(*

.. <legal notes>

legal notes
=================
| SPDX-FileCopyrightText: © 2026 Oleksandr Tiutyk <trofimich@gmail.com>
| SPDX-License-Identifier: LGPL-3.0-only
| For details check: LGPL-3.0-only_

.. _LGPL-3.0-only: https://www.gnu.org/licenses/lgpl-3.0.en.html

.. </legal notes>

*)

{attribute 'no_explicit_call' := 'do not call this function block directly'} 
FUNCTION_BLOCK AdsLogger EXTENDS Object IMPLEMENTS ILogger
VAR
	_ClassName : STRING := __POUNAME();
END_VAR

{attribute 'monitoring' := 'call'}
PROPERTY ClassName : REFERENCE TO STRING
GET
ClassName REF= _ClassName;
END_GET
END_PROPERTY

METHOD Execute
// nothing to do for ADS logger
END_METHOD

{attribute 'monitoring' := 'call'}
PROPERTY NamespaceName : STRING
GET
NamespaceName := CurrentNamespace.Name;
END_GET
END_PROPERTY

{attribute 'monitoring' := 'call'}
PROPERTY SelfSize : ULINT
GET
SelfSize := XSIZEOF(THIS^);
END_GET
END_PROPERTY

METHOD TryLogError : BOOL
VAR_INPUT
	error : REFERENCE TO ERROR;
	messageNumber : REFERENCE TO ULINT := 0;
END_VAR
VAR
	message : ERROR_MESSAGE;
END_VAR
IF NOT __ISVALIDREF(error) THEN
	RETURN;
END_IF

message := error.ToString(ERROR_SOURCE_DISPLAY_MODE.TOP_AND_ROOT, TIMESTAMP_DISPLAY_MODE.LOCAL);

TryLogError := TryLogMessage(SEL(error.Severity = ERROR_SEVERITY.CRITICAL, LOG_CATEGORY.ERROR, LOG_CATEGORY.CRITICAL_ERROR), message, messageNumber);
END_METHOD

METHOD TryLogException : BOOL
VAR_INPUT
	exception : IException;
	severity : ERROR_SEVERITY;
	messageNumber : REFERENCE TO ULINT := 0;
END_VAR
VAR
	message : ERROR_MESSAGE;
	aggregateException : IAggregateException;
	innerException : IException;
	i : DINT;
END_VAR
IF exception = 0 THEN
	RETURN;
END_IF

IF NOT __QUERYINTERFACE(exception, aggregateException) OR_ELSE aggregateException.InnerExceptionCount = 0 THEN
	message := exception.GetMessage(TRUE, TIMESTAMP_DISPLAY_MODE.LOCAL);
	
	TryLogException := TryLogMessage(SEL(severity = ERROR_SEVERITY.CRITICAL, LOG_CATEGORY.ERROR, LOG_CATEGORY.CRITICAL_ERROR), message, messageNumber);
ELSE
	IF aggregateException.InnerExceptionCount > 1 THEN
		// reverce order
		TryLogException := TryLogMessage(LOG_CATEGORY.ERROR, "<<< aggregate exception end <<<");
		
		FOR i := TO_DINT(aggregateException.InnerExceptionCount) - 1 TO 0 BY -1 DO
			innerException := aggregateException.GetInnerException(i);
			
			message := WideStrings.Concat255("  ", innerException.GetMessage(TRUE, TIMESTAMP_DISPLAY_MODE.LOCAL));
			
			TryLogException := TryLogException AND TryLogMessage(SEL(severity = ERROR_SEVERITY.CRITICAL, LOG_CATEGORY.ERROR, LOG_CATEGORY.CRITICAL_ERROR), message);		
		END_FOR
		
		TryLogException := TryLogException AND TryLogMessage(SEL(severity = ERROR_SEVERITY.CRITICAL, LOG_CATEGORY.ERROR, LOG_CATEGORY.CRITICAL_ERROR), ">>> aggregate exception start >>>", messageNumber);
	ELSE		
		innerException := aggregateException.GetInnerException(0);
		
		message := innerException.GetMessage(TRUE, TIMESTAMP_DISPLAY_MODE.LOCAL);
		
		TryLogException := TryLogMessage(SEL(severity = ERROR_SEVERITY.CRITICAL, LOG_CATEGORY.ERROR, LOG_CATEGORY.CRITICAL_ERROR), message);
	END_IF
END_IF
END_METHOD

METHOD TryLogMessage : BOOL
VAR_INPUT
	category : LOG_CATEGORY;	
END_VAR
VAR_IN_OUT CONSTANT
	message : ERROR_MESSAGE;
END_VAR
VAR_INPUT
	messageNumber : REFERENCE TO ULINT := 0;
END_VAR
VAR
	messageControlMask : DWORD;
END_VAR
CASE category OF
	LOG_CATEGORY.DEBUG, LOG_CATEGORY.INFORMATION:
		messageControlMask := Tc2_System.Global_Variables.ADSLOG_MSGTYPE_LOG;
		
	LOG_CATEGORY.WARNING:
		messageControlMask := Tc2_System.Global_Variables.ADSLOG_MSGTYPE_WARN;
	
	LOG_CATEGORY.ERROR, LOG_CATEGORY.CRITICAL_ERROR:
		messageControlMask := Tc2_System.Global_Variables.ADSLOG_MSGTYPE_ERROR;
END_CASE

IF __ISVALIDREF(messageNumber) THEN
	TryLogMessage := Tc2_System.ADSLOGSTR(
		msgCtrlMask := messageControlMask, 
		msgFmtStr := Strings.Concat255(TO_STRING(Exceptions.MESSAGE_NUMBER_PREFIX), Exceptions.LOG_CATEGORY_PREFIXES[category], TO_STRING(messageNumber), TO_STRING(Exceptions.MESSAGE_NUMBER_SUFFIX), TO_STRING(message)), 
		strArg := '') = 0;
ELSE
	TryLogMessage := Tc2_System.ADSLOGSTR(msgCtrlMask := messageControlMask, msgFmtStr := TO_STRING(message), strArg := '') = 0;
END_IF
END_METHOD

END_FUNCTION_BLOCK

(* stored: Version 1.1.0.1
   POU AdsLogger: Id {c95de8ac-0505-4250-b81e-2b0cbe2bb2ed}, SpecialFunc None
   Property ClassName: Id {c900fbb9-86d0-4a3f-9595-f30e1df1d1f1}
   Get Get: Id {910140d1-6146-4f27-82a4-105ab45c7077}
   Method Execute: Id {7f679376-d6c2-4628-9f18-706629e6a200}
   Property NamespaceName: Id {c38469fc-4ff8-41a9-b499-75e413a00bb3}
   Get Get: Id {bcccda69-31bf-4d44-868c-2415428102e1}
   Property SelfSize: Id {c266c68f-d111-413c-997b-ce427475c7b9}
   Get Get: Id {368ffd0e-de98-47d3-99fe-4d83a0af5f22}
   Method TryLogError: Id {20bf6186-2dc6-4029-8680-18c8f237e377}
   Method TryLogException: Id {52444f42-e6c7-4828-baa7-3f12fe45268b}
   Method TryLogMessage: Id {936430cf-8fdd-47d1-875f-690550891879} *)
